(* Logix 5000 project; controller EuniceF_Lab1 vendor 1 type 14 code 150 rev 37.11; software revision 37.00 *)

TASK MainTask (continuous, watchdog 500 ms) : MainProgram

MODULES
   Local : vendor 1 type 14 code 150 (Compact 0, rev 37.11)
      Discrete_IO : Embedded (Compact 1, rev 3.1, Output RPI 20 ms)
      Analog_IO : Embedded (Compact 2, rev 1.1, Output RPI 80 ms)
      Counters : Embedded (Compact 3, rev 1.1, Output RPI 20 ms)
END_MODULES

VAR_GLOBAL   (* controller tags *)
   CloseTime : STRING;
   ContinueMess : STRING;
   Countfor60cm : DINT;
   Default_Kfactor : DINT;
   Diif_Pressure : ALIAS FOR Local:2:I.Ch3Data;
   Done : ALIAS FOR Local:1:I.Data.15;
   Drain_Manual : ALIAS FOR Local:1:I.Data.4;
   DrainClose : DINT;
   DrainValve : ALIAS FOR Local:1:O.Data.10;
   Fill_Valve : ALIAS FOR Local:2:I.Ch3Data;
   Full : INT := 29208;
   Full_Btn : ALIAS FOR Local:1:I.Data.13;
   Good : ALIAS FOR Local:1:I.Data.14;
   Half : INT := -288;
   Half_Btn : ALIAS FOR Local:1:I.Data.12;
   HSC1_CurentCount : ALIAS FOR Local:3:I.Ctr0CurrentCount;
   HSCMessage : STRING;
   K_factor : DINT;
   KfactorMessage : STRING;
   LevelMax : DINT;
   LevelMin : DINT;
   MainMessage : STRING;
   Mixer : ALIAS FOR Local:1:O.Data.9;
   Prove : ALIAS FOR Local:1:I.Data.7;
   provebMessage : STRING;
   ProveMess : STRING;
   Pump : ALIAS FOR Local:1:O.Data.8;
   PumpButton : STRING;
   PumpMessage : STRING;
   Quarter : INT := -15037;
   Quarter_Btn : ALIAS FOR Local:1:I.Data.11;
   Reset_HSC : ALIAS FOR Local:3:O.Ctr0SoftPreset;
   SEQ : DINT;
   Start : ALIAS FOR Local:1:I.Data.1;
   StartButton : STRING;
   StartMessage : STRING;
   Status : STRING;
   Stop : ALIAS FOR Local:1:I.Data.2;
   Stop_Emergency : STRING;
   Stop_MainMessage : STRING;
   Stopbutton : STRING;
   StopPressed : STRING;
   T1 : TIMER;
   Time : TIMER;
   TimerDrain : DINT;
   Valve_Position : ALIAS FOR Local:2:O.Ch1Data;
   valveMess : STRING;
   ValveTime : STRING;
   Zero : ALIAS FOR Local:1:I.Data.3;
END_VAR

PROGRAM MainProgram   (* main routine MainRoutine *)
VAR
   TimeDrain : TIMER;
   TimeEndDrain : TIMER;
END_VAR

ROUTINE MainRoutine   (* ladder *)
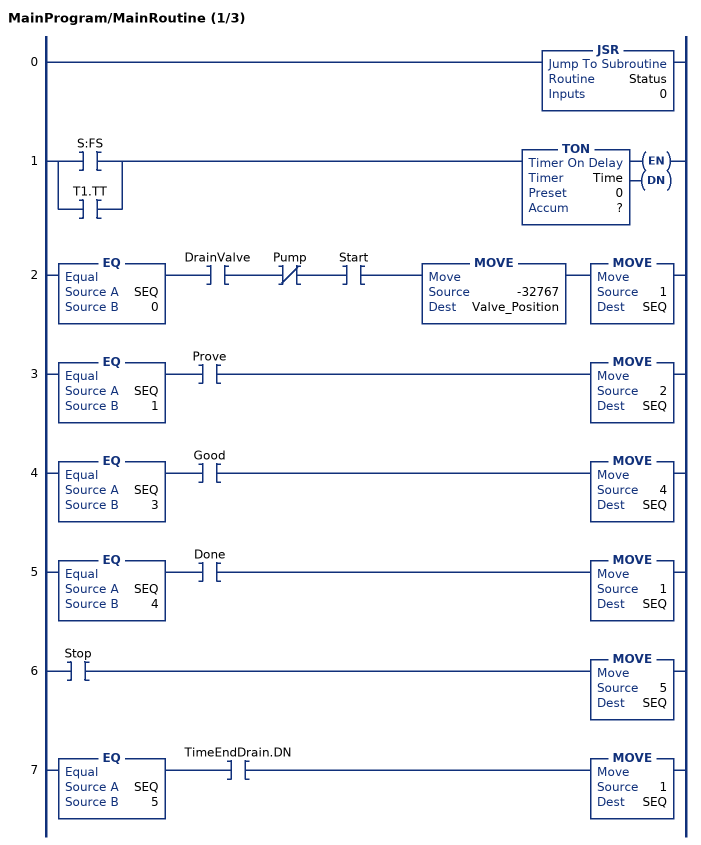
   0: JSR(Status,0);
   1: [XIC(S:FS) ,XIC(T1.TT) ]TON(Time,?,?);
   2: EQ(SEQ,0)XIC(DrainValve)XIO(Pump)XIC(Start)MOVE(-32767,Valve_Position)MOVE(1,SEQ);
   3: EQ(SEQ,1)XIC(Prove)MOVE(2,SEQ);
   4: EQ(SEQ,3)XIC(Good)MOVE(4,SEQ);
   5: EQ(SEQ,4)XIC(Done)MOVE(1,SEQ);
   6: XIC(Stop)MOVE(5,SEQ);
   7: EQ(SEQ,5)XIC(TimeEndDrain.DN)MOVE(1,SEQ);
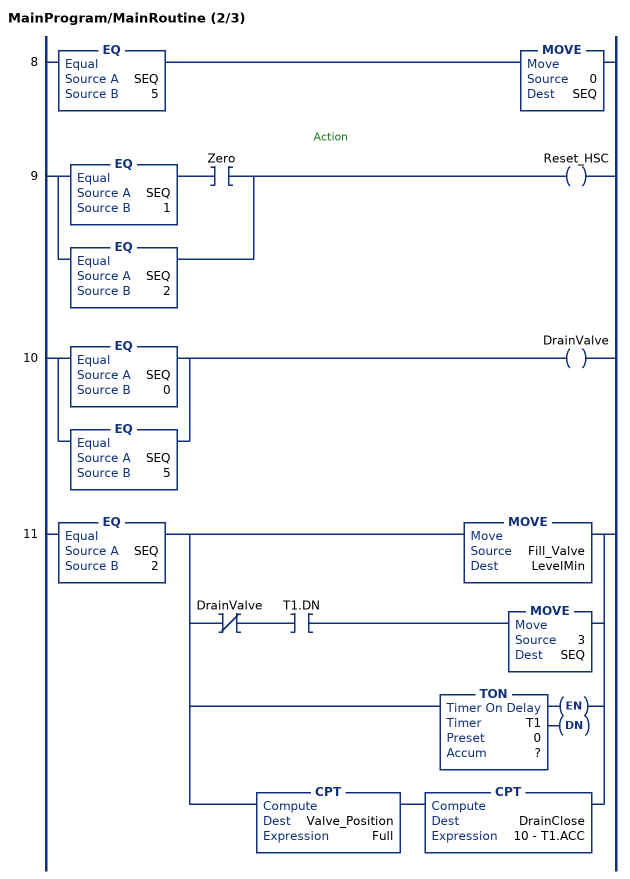
   8: EQ(SEQ,5)MOVE(0,SEQ);
   // Action
   9: [EQ(SEQ,1) XIC(Zero) ,EQ(SEQ,2) ]OTE(Reset_HSC);
   10: [EQ(SEQ,0) ,EQ(SEQ,5) ]OTE(DrainValve);
   11: EQ(SEQ,2)[MOVE(Fill_Valve,LevelMin) ,XIO(DrainValve) XIC(T1.DN) MOVE(3,SEQ) ,TON(T1,?,?) ,CPT(Valve_Position,Full) CPT(DrainClose,10 - T1.ACC) ];
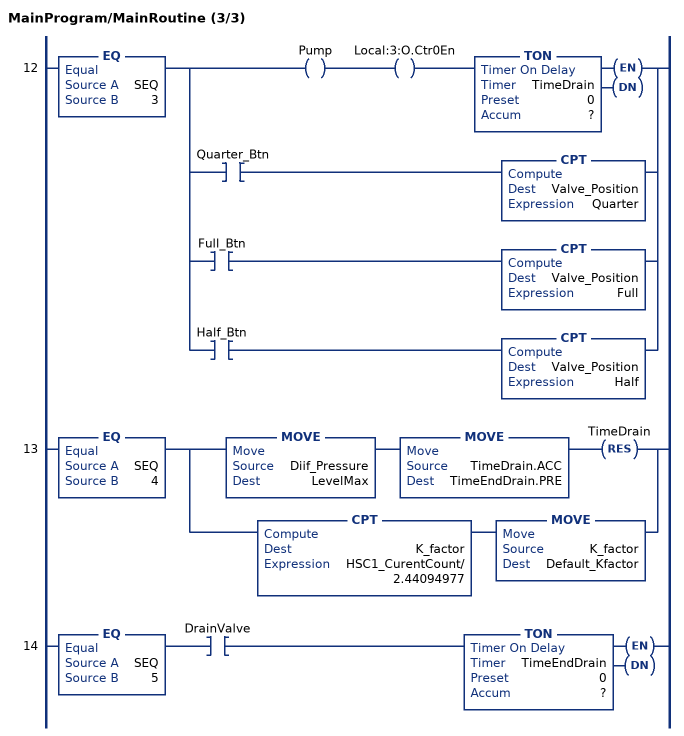
   12: EQ(SEQ,3)[OTE(Pump) OTE(Local:3:O.Ctr0En) TON(TimeDrain,?,?) ,XIC(Quarter_Btn) CPT(Valve_Position,Quarter) ,XIC(Full_Btn) CPT(Valve_Position,Full) ,XIC(Half_Btn) CPT(Valve_Position,Half) ];
   13: EQ(SEQ,4)[MOVE(Diif_Pressure,LevelMax) MOVE(TimeDrain.ACC,TimeEndDrain.PRE) RES(TimeDrain) ,CPT(K_factor,HSC1_CurentCount/ 2.44094977) MOVE(K_factor,Default_Kfactor) ];
   14: EQ(SEQ,5)XIC(DrainValve)TON(TimeEndDrain,?,?);
END_ROUTINE

ROUTINE Status   (* structured text *)
   if SEQ=0 then
   	concat(StartMessage,StartButton,MainMessage);
   
   end_if;
   if SEQ=1 then
   	concat(provebMessage,ProveMess,MainMessage);
   	concat(Stop_Emergency,Stopbutton,Stop_MainMessage);
   end_if;
   
   if SEQ=2 then
   	DTOS(DrainClose,CloseTime);
   	concat(ValveTime,CloseTime,MainMessage);
   	concat(Stop_Emergency,Stopbutton,Stop_MainMessage);
   end_if;
   
   if SEQ=3 then
   	DTOS(HSC1_CurentCount,HSCMessage);
   	concat(HSCMessage,PumpButton,MainMessage);
   	concat(Stop_Emergency,Stopbutton,Stop_MainMessage);
   end_if;
   
   if SEQ=4 then
   	DTOS(K_factor,KfactorMessage);
   	concat(KfactorMessage,ContinueMess,MainMessage);
   	concat(Stop_Emergency,Stopbutton,Stop_MainMessage);
   end_if;
   if SEQ=5 then
   	concat(Stop_Emergency,Stopbutton,Stop_MainMessage);
   end_if;
   
   
   
END_ROUTINE
END_PROGRAM
